// TIA Portal V16 export
// export: Created 2021-11-12T13:33:07.9327842Z, ExportSetting WithDefaults, DisplayName Totally Integrated Automation Portal, DisplayVersion V16 Update 3, DisplayName TIA Portal Version Control Interface, DisplayVersion V16 Update 2, DisplayName TIA Portal Openness, DisplayVersion V16 Update 3, DisplayName SINAMICS Startdrive Advanced, DisplayVersion V16 Update 5, DisplayName SINAMICS Startdrive G130, G150, S120, S150, SINAMICS MV, S210, DisplayVersion V16 Update 5, DisplayName SINAMICS Startdrive G110M, G120, G120C, G120D, G120P, G115D, DisplayVersion V16 Update 5, DisplayName STEP 7 Professional, DisplayVersion V16 Update 3, DisplayName STEP 7 Safety, DisplayVersion V16, DisplayName WinCC UA Professional, DisplayVersion V16 Update 3
DATA_BLOCK "IDB_IM_410+UH31+KF10"   // DB219
{ DB_Accessible_From_OPC_UA := 'FALSE' }
VERSION : 0.1
// stored: AutoNumber true, DBAccessibleFromOPCUA false, InstanceOfName IM_410+UH31+KF10, InstanceOfType FB
"IM_410+UH31+KF10"
   // VAR
   //    KF11_Ix0 : "STD_CH_DI";
   //    KF11_Ix1 { S7_SetPoint := 'True'} : "STD_CH_DI";
   //    KF11_Ix2 { S7_SetPoint := 'True'} : "STD_CH_DI";
   //    KF11_Ix3 { S7_SetPoint := 'True'} : "STD_CH_DI";
   //    KF11_Ix4 { S7_SetPoint := 'True'} : "STD_CH_DI";
   //    KF11_Ix5 { S7_SetPoint := 'True'} : "STD_CH_DI";
   //    KF11_Ix6 { S7_SetPoint := 'True'} : "STD_CH_DI";
   //    KF11_Ix7 { S7_SetPoint := 'True'} : "STD_CH_DI";
   //    KF12_Ix0 { S7_SetPoint := 'True'} : "STD_CH_DI";
   //    KF12_Ix1 { S7_SetPoint := 'True'} : "STD_CH_DI";
   //    KF12_Ix2 { S7_SetPoint := 'True'} : "STD_CH_DI";
   //    KF12_Ix3 { S7_SetPoint := 'True'} : "STD_CH_DI";
   //    KF12_Ix4 { S7_SetPoint := 'True'} : "STD_CH_DI";
   //    KF12_Ix5 { S7_SetPoint := 'True'} : "STD_CH_DI";
   //    KF12_Ix6 { S7_SetPoint := 'True'} : "STD_CH_DI";
   //    KF12_Ix7 { S7_SetPoint := 'True'} : "STD_CH_DI";
   //    KF51_AI0 { S7_SetPoint := 'True'} : "STD_CH_AI";
   //    KF51_AI1 { S7_SetPoint := 'True'} : "STD_CH_AI";
   //    KF52_AI0 { S7_SetPoint := 'True'} : "STD_CH_AI";
   //    KF52_AI1 { S7_SetPoint := 'True'} : "STD_CH_AI";
   // END_VAR
BEGIN
END_DATA_BLOCK
